RoboDK station: dofbot_DX_6_axis_generic_final_add_blcok_V1.0.0.rdk

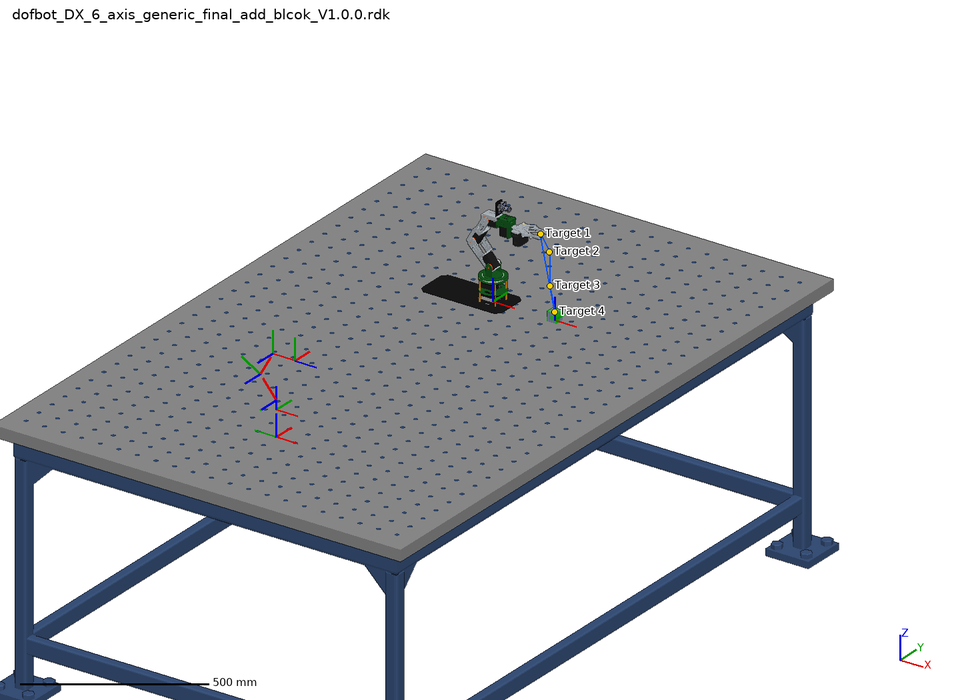
[picture v0: the station drawn from its stored meshes, robots at their saved joint values, targets as dots, program paths as lines]
Station dofbot_DX_6_axis_generic_final_add_blcok_V1.0.0 (saved by RoboDK 6.0.3). Poses are relative to the parent item; angles as X-Y-Z fixed-axis rotations.
  - frame Frame 1 at (0, 0, 0) mm
    - object dofbot_BASE_FRAME_add_axis at (0, 0, 0) mm, size 367.1 x 120 x 302.4 mm, geometry from dofbot_BASE_FRAME_add_axis.STEP
    - frame Frame 2 at (0, 0, 80) mm
      - object dofbot_LINK_1_add_axis at (0, 0, 0) mm, size 60.9 x 54.8 x 86.3 mm, geometry from dofbot_LINK_1_add_axis.STEP
        - frame Frame 3 at (0, 0, 27.5) mm, rotated rx -90 ry -50 rz 180 deg
          - object dofbot_LINK_2_add_axis at (0, 0, 0) mm, size 106.7 x 29.1 x 42.7 mm, geometry from dofbot_LINK_2_add_axis.STEP
          - frame Frame 4 at (82.85, 0, 0) mm, rotated rx 0 ry 0 rz -70 deg
            - object dofbot_LINK_3_add_axis at (0, 0, 0) mm, size 106.7 x 29.1 x 42.7 mm, geometry from dofbot_LINK_3_add_axis.STEP
            - frame Frame 5 at (82.85, 0, 0) mm, rotated rx 0 ry 0 rz -60 deg
              - object dofbot_LINK_4_add_axis at (0, 0, 0) mm, size 88 x 50 x 38.7 mm, geometry from dofbot_LINK_4_add_axis.STEP
              - frame Frame 6 at (70, -2.5, -1) mm, rotated rx 0 ry 90 rz 0 deg
                - object dofbot_LINK_5_add_axis at (0, 0, 0) mm, size 22.9 x 44 x 35.1 mm, geometry from dofbot_LINK_5_add_axis.STEP
                  - frame Frame 7 at (0, 0, 0) mm
                    - object dofbot_LINK_6_add_axis at (0, 0, 0) mm, size 62.7 x 55.3 x 110.3 mm, geometry from dofbot_LINK_6_add_axis.STEP
  - frame My Mechanism Base at (0, 1000, 0) mm
    - robot My Mechanism: 6 axes
        modified DH rows (alpha deg, a mm, theta deg, d mm): 0, 0, 0, 107.5; 90, 0, 130, 0; 0, 82.85, -70, 0; 0, 82.85, -60, 0; -90, 70, -90, 0; -90, 0, 0, 95
        joint limits [-200, -200, -200, -200, 0, -200] to [200, 200, 200, 200, 0, 200]; home [0, 0, 0, 0, 0, 0]; saved at [0, 0, 0, 0, 0, 0]
      - tool Tool 1, TCP at (0, 0, 0) mm
  - frame Frame 9 at (0, 0, 0) mm, rotated rx 0 ry 0 rz 90 deg
    - object Table 2000x1200x800mm at (0, 0, 0) mm, size 2020 x 1340 x 800 mm, geometry from Table-2000x1200x800mm.sld
    - target Target 1 (Cartesian target) at (1000, -153.17, 242.72) mm, rotated rx -90 ry 0 rz -180 deg; joints [0, 0, 0, 0, 0, 0] of My Mechanism
    - target Target 2 (Cartesian target) at (1000, -183.19, 197.99) mm, rotated rx -105.15 ry 0 rz -180 deg; joints [0, -15.15, 0, 0, 0, 0] of My Mechanism
    - target Target 3 (Cartesian target) at (1000, -184.15, 97.59) mm, rotated rx -134.28 ry 0 rz -180 deg; joints [0, -30.68, -12.82, -0.78, 0, 0] of My Mechanism
    - target Target 4 (Cartesian target) at (1000, -199.54, 24.67) mm, rotated rx -153.68 ry 0 rz -180 deg; joints [0, -71.84, 8.16, 0, 0, 0] of My Mechanism
  - frame Frame 10 at (200, 1000, 0) mm
    - object block_green_3by3 at (0, 0, 0) mm, rotated rx 0 ry 0 rz 90 deg, size 30 x 30 x 30 mm, geometry from block_green_3by3.STEP
  - program Prog1 (1 instructions, listed below)
  - program Prog2 (6 instructions, listed below)
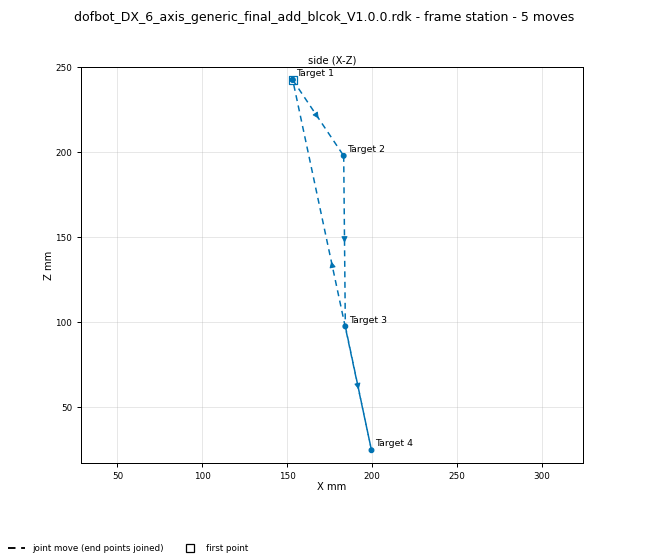
[picture p0: tool path of dofbot_DX_6_axis_generic_final_add_blcok_V1.0.0.rdk in frame station, 5 of 5 moves have a stored position in this frame; points joined in program order, loops and branches not executed]

--- program Prog1 (robot My Mechanism) ---
  Set Ref.: Frame 9

--- program Prog2 (robot My Mechanism) ---
  Set Ref.: Frame 9
  MoveJ (Target 1)
  MoveJ (Target 2)
  MoveJ (Target 3)
  MoveJ (Target 4)
  MoveJ (Target 1)
